// TIA Portal project "SORTIROZO_GEP_VEZERLES" (V15)

(* hardware
DEVICE "S71500/ET200MP-Station_1"  S7-1500 station
   slot 0: "Profilschiene_0"  6ES7 590-1***0-0AA0
   slot 1: "PLC_1"  CPU 1511-1 PN  6ES7 511-1AK00-0AB0  V1.8
   slot 2: "AI 8xU/I/RTD/TC ST_1"  AI 8xU/I/RTD/TC ST  6ES7 531-7KF00-0AB0  V2.0
   slot 3: "AI 8xU/I/RTD/TC ST_2"  AI 8xU/I/RTD/TC ST  6ES7 531-7KF00-0AB0  V2.0
   slot 4: "AI 8xU/I/RTD/TC ST_3"  AI 8xU/I/RTD/TC ST  6ES7 531-7KF00-0AB0  V2.0
   slot 5: "AI 8xU/I/RTD/TC ST_4"  AI 8xU/I/RTD/TC ST  6ES7 531-7KF00-0AB0  V2.0
   slot 6: "DI 16x24VDC BA_1"  DI 16x24VDC BA  6ES7 521-1BH10-0AA0  V1.0
*)

// ===== PLC "PLC_1"  CPU 1511-1 PN =====

VAR_GLOBAL   // PLC tag table "Standard-Variablentabelle"
   "System_Byte" AT %MB1 : Byte;
   "FirstScan" AT %M1.0 : Bool;
   "DiagStatusUpdate" AT %M1.1 : Bool;
   "AlwaysTRUE" AT %M1.2 : Bool;
   "AlwaysFALSE" AT %M1.3 : Bool;
   "Clock_Byte" AT %MB0 : Byte;
   "Clock_10Hz" AT %M0.0 : Bool;
   "Clock_5Hz" AT %M0.1 : Bool;
   "Clock_2.5Hz" AT %M0.2 : Bool;
   "Clock_2Hz" AT %M0.3 : Bool;
   "Clock_1.25Hz" AT %M0.4 : Bool;
   "Clock_1Hz" AT %M0.5 : Bool;
   "Clock_0.625Hz" AT %M0.6 : Bool;
   "Clock_0.5Hz" AT %M0.7 : Bool;
END_VAR

VAR_GLOBAL   // PLC tag table "IO"
   "PART_SENSOR_BIT_0" AT %I0.0 : Bool;
   "PART_SENSOR_BIT_1" AT %I0.1 : Bool;
   "PART_SENSOR_BIT_2" AT %I0.2 : Bool;
   "PART_SENSOR_BIT_3" AT %I0.3 : Bool;
   "PART_CAPACITIVE_SENSOR" AT %I0.4 : Bool;
   "PART_INDUCTIVE_SENSOR" AT %I0.5 : Bool;
   "REFLECTIVE_SENSOR" AT %I0.6 : Bool;
   "MANUAL_SWITCH" AT %I0.7 : Bool;
   "AUTO_SWITCH" AT %I1.0 : Bool;
   "START_BUTTON" AT %I1.1 : Bool;
   "STOP_BUTTON" AT %I1.2 : Bool;
   "ROBOT_PART_PLACE_GRAB_DEDECTED" AT %I1.3 : Bool;
   "ROBOT_PART_PLACE_X_IS_MOVING" AT %I1.4 : Bool;
   "ROBOT_PART_PLACE_Z_IS_MOVING" AT %I1.5 : Bool;
   "ROBOT_PART_PLACE_IS_ROTATING" AT %I1.6 : Bool;
   "ROBOT_PART_PICK_GRAB_DEDECTED" AT %I1.7 : Bool;
   "ROBOT_PART_PICK_X_IS_MOVING" AT %I2.0 : Bool;
   "ROBOT_PART_PICK_Z_IS_MOVING" AT %I2.1 : Bool;
   "ROBOT_PART_PICK_IS_ROTATING" AT %I2.2 : Bool;
   "STACK_LIGHT_RED" AT %Q0.0 : Bool;
   "STACK_LIGHT_GREEN" AT %Q0.1 : Bool;
   "STACK_LIGHT_YELLOW" AT %Q0.2 : Bool;
   "START_BUTTON_LIGHT" AT %Q0.3 : Bool;
   "STOP_BUTTON_LIGHT" AT %Q0.4 : Bool;
   "PART_INSPECT_STOP_BLADE" AT %Q0.5 : Bool;
   "PART_PICKUP_STOP_BLADE" AT %Q0.6 : Bool;
   "ROBOT_PART_PLACE_X" AT %Q0.7 : Bool;
   "ROBOT_PART_PLACE_Z" AT %Q1.0 : Bool;
   "ROBOT_PART_PLACE_GRAB" AT %Q1.1 : Bool;
   "ROBOT_PART_PLACE_ROTATE_CW" AT %Q1.2 : Bool;
   "ROBOT_PART_PLACE_ROTATE_CCW" AT %Q1.3 : Bool;
   "ROBOT_PART_PICK_X" AT %Q1.4 : Bool;
   "ROBOT_PART_PICK_Z" AT %Q1.5 : Bool;
   "ROBOT_PART_PICK_GRAB" AT %Q1.6 : Bool;
   "ROBOT_PART_PICK_ROTATE_CW" AT %Q1.7 : Bool;
   "ROBOT_PART_PICK_ROTATE_CCW" AT %Q2.0 : Bool;
   "PART_CONVEYOR" AT %Q2.1 : Bool;
END_VAR

DATA_BLOCK "mainProgram_DB"   // DB1
{ S7_Optimized_Access := 'TRUE' }
VERSION : 0.1
// stored: InstanceOfName mainProgram
"mainProgram"
BEGIN
END_DATA_BLOCK

DATA_BLOCK "mainProgram_DB_1"   // DB5
{ S7_Optimized_Access := 'TRUE' }
VERSION : 0.1
// stored: InstanceOfName mainProgram
"mainProgram"
BEGIN
END_DATA_BLOCK

// folder: System blocks/Program resources

DATA_BLOCK "IEC_Timer_0_DB"   // DB10
{ S7_Optimized_Access := 'TRUE' }
AUTHOR : Simatic
FAMILY : IEC
NAME : IEC_TMR
VERSION : 1.0
// stored: InstanceOfName IEC_TIMER
"IEC_TIMER"
BEGIN
END_DATA_BLOCK

// folder: (top level)

FUNCTION_BLOCK "mainProgram"   // FB1, SCL
{ S7_Optimized_Access := 'TRUE' }
VERSION : 0.1
   VAR_INPUT
      partSensorBit0 : Bool;
      partSensorBit1 : Bool;
      partSensorBit2 : Bool;
      partSensorBit3 : Bool;
      partCapacitiveSensor : Bool;
      partInductiveSensor : Bool;
      partReflectiveSensor : Bool;
      manualSwitch : Bool;
      autoSwitch : Bool;
      startButton : Bool;
      stopButton : Bool;
      robotPartPlaceGrabDedected : Bool;
      robotPartPlaceXIsMoving : Bool;
      robotPartPlaceZIsMoving : Bool;
      robotPartPlaceIsRotating : Bool;
      robotPartPickIsDedected : Bool;
      robotPartPickXIsMoving : Bool;
      robotPartPickZIsMoving : Bool;
      robotPartPickIsRotating : Bool;
   END_VAR
   VAR_OUTPUT
      stackLightRed : Bool;
      stackLightGreen : Bool;
      stackLightYellow : Bool;
      startButtonLighgt : Bool;
      stopButtonLight : Bool;
      partInspectStopBlade : Bool;
      partPickupStopBlade : Bool;
      robotPartPlaceX : Bool;
      robotPartPlaceZ : Bool;
      robotPartPlaceGrab : Bool;
      robotPartPlaceRotateCW : Bool;
      robotPartPlaceRotateCCW : Bool;
      robotPartPickX : Bool;
      robotPartPickZ : Bool;
      robotPartPickGrab : Bool;
      robotPartPickRotateCW : Bool;
      robotPartPickRotateCCW : Bool;
      partConveyor : Bool;
   END_VAR
   VAR
      robotRotateCounter : Int;
      "timer" : Time;
      onDelayCheck : Bool;
      fallingEgdeDedect : Bool;
      risingEgdeDedect : Bool;
      deviceState : Int;
      pickUpRobotState : Int;
      partPlaceRobotState : Int;
      cameraControlState : Int;
      partCameraData : Int;
      conveyorControlState : Int;
   END_VAR
   VAR CONSTANT
      CONVEYOR_MOVING_GRAY : Time := T#10s;
      CONVEYOR_MOVING_BLUE : Time := T#6s;
      ROBOT_PICK_NEXT_STEP_WAIT_TIME : Time := T#1s;
      STATE_INIT : Int;
      STATE_WAIT_FOR_START : Int := 1;
      STATE_IDLE : Int := 3;
      STATE_ROBOT_PICK_IDLE : Int;
      STATE_ROBOT_PICK_MOVE_PART_X : Int := 2;
      STATE_ROBOT_PICK_MOVE_PART_Z : Int := 3;
      STATE_ROBOT_PICK_GRAB_PART : Int := 4;
      STATE_ROBOT_PICK_ROTATE_TO_CONVEYER : Int := 7;
      STATE_ROBOT_PICK_PLACE_PART : Int := 8;
      STATE_ROBOT_PICK_CHECK_FOR_BASE_POSITION : Int := 9;
      STATE_CAMERA_IDLE : Int;
      STATE_CAMERA_READ_PRODUCT_DATA : Int := 1;
      STATE_CONVEYOR_IDLE : Int;
      STATE_CONVEYOR_GRAY : Int := 1;
      STATE_CONVEYOR_BLUE : Int := 2;
      STATE_CONVEYOR_GREEN : Int := 3;
      STATE_PART_PLACE_ROBOT_IDLE : Int;
      STATE_PART_PLACE_ROBOT_MOVE_X : Int := 1;
      STATE_PART_PLACE_ROBOT_MOVE_Z : Int := 2;
      STATE_PART_PLACE_ROBOT_GRAB : Int := 3;
      STATE_PART_PLACE_ROBOT_ROTATE_TO_CONVEYER : Int := 4;
      STATE_PART_PLACE_ROBOT_PLACE_PART : Int := 5;
   END_VAR
BEGIN
   CASE #deviceState OF
       #STATE_INIT:
           #stackLightYellow := "Clock_2Hz";
           #partInspectStopBlade := TRUE;
           #partPickupStopBlade := TRUE;
           #robotPartPlaceRotateCW := TRUE;

           "F_TRIG_DB"(CLK:=#robotPartPlaceIsRotating,
                       Q=>#fallingEgdeDedect);

           IF #fallingEgdeDedect THEN
               #stackLightYellow := FALSE;
               #stackLightRed := TRUE;
               #deviceState := #STATE_WAIT_FOR_START;
           END_IF;

       #STATE_WAIT_FOR_START:
           "R_TRIG_DB"(CLK:=#startButton,
                       Q=>#risingEgdeDedect);

           IF #risingEgdeDedect THEN
               #deviceState := #STATE_IDLE;
               #pickUpRobotState := #STATE_ROBOT_PICK_MOVE_PART_X;
           END_IF;
   END_CASE;

   CASE #pickUpRobotState OF
       #STATE_ROBOT_PICK_MOVE_PART_X:
           #robotPartPickX := TRUE;

           "F_TRIG_DB_1"(CLK:=#robotPartPickXIsMoving,
                         Q=>#fallingEgdeDedect);

           IF #fallingEgdeDedect THEN
               #pickUpRobotState := #STATE_ROBOT_PICK_MOVE_PART_Z;
           END_IF;

       #STATE_ROBOT_PICK_MOVE_PART_Z:
           #robotPartPickZ := TRUE;

           "F_TRIG_DB_2"(CLK:=#robotPartPickZIsMoving,
                         Q=>#fallingEgdeDedect);

           IF #fallingEgdeDedect THEN
               WAIT(WT := 10000);
               #robotPartPickGrab := TRUE;
               #stackLightRed := FALSE;
               #pickUpRobotState := #STATE_ROBOT_PICK_GRAB_PART;
           END_IF;

       #STATE_ROBOT_PICK_GRAB_PART:
           #robotPartPickGrab := TRUE;

           IF #robotPartPickIsDedected THEN
               WAIT(WT := 1000);
               #robotPartPickZ := FALSE;
               #pickUpRobotState := #STATE_ROBOT_PICK_ROTATE_TO_CONVEYER;
           END_IF;

       #STATE_ROBOT_PICK_ROTATE_TO_CONVEYER:
           #robotPartPickRotateCCW := TRUE;

           "F_TRIG_DB_3"(CLK:=#robotPartPickIsRotating,
                         Q=>#fallingEgdeDedect);

           IF #fallingEgdeDedect THEN
               WAIT(WT := 10000);
               #robotPartPickRotateCCW := FALSE;
               #pickUpRobotState := #STATE_ROBOT_PICK_PLACE_PART;
           END_IF;

       #STATE_ROBOT_PICK_PLACE_PART:
           #robotPartPickZ := TRUE;

           "F_TRIG_DB_2"(CLK := #robotPartPickZIsMoving,
                         Q => #fallingEgdeDedect);

           IF #fallingEgdeDedect THEN
               WAIT(WT := 10000);
               #robotPartPickGrab := FALSE;
               #robotPartPickZ := FALSE;
               #robotPartPickX := FALSE;
               #robotPartPickRotateCW := TRUE;
               #pickUpRobotState := #STATE_ROBOT_PICK_CHECK_FOR_BASE_POSITION;
               #cameraControlState := #STATE_CAMERA_READ_PRODUCT_DATA;
           END_IF;

   END_CASE;

   CASE #cameraControlState OF
       #STATE_CAMERA_READ_PRODUCT_DATA:
           IF #partSensorBit0 = TRUE AND #partSensorBit3 = TRUE THEN
               #conveyorControlState := #STATE_CONVEYOR_GRAY;
               #cameraControlState := #STATE_CAMERA_IDLE;
           END_IF;

           IF #partSensorBit0 = TRUE AND #partSensorBit1 = TRUE THEN
               #conveyorControlState := #STATE_CONVEYOR_BLUE;
               #cameraControlState := #STATE_CAMERA_IDLE;
           END_IF;

           IF #partSensorBit1 = TRUE AND #partSensorBit2 = TRUE THEN
               #conveyorControlState := #STATE_CONVEYOR_GREEN;
               #cameraControlState := #STATE_CAMERA_IDLE;
           END_IF;
   END_CASE;

   CASE #conveyorControlState OF
       #STATE_CONVEYOR_GRAY:
           #partConveyor := TRUE;
           #partInspectStopBlade := FALSE;
           #partPickupStopBlade := FALSE;

           "IEC_Timer_0_DB".TON(IN:=TRUE,
                                PT:=#CONVEYOR_MOVING_GRAY,
                                Q=>#onDelayCheck,
                                ET=>#timer);

           IF #onDelayCheck THEN
               #robotPartPickRotateCW := FALSE;
               #conveyorControlState := #STATE_CONVEYOR_IDLE;
               #partConveyor := FALSE;
               "IEC_Timer_0_DB".TON(IN := FALSE,
                                    PT := #CONVEYOR_MOVING_GRAY,
                                    Q => #onDelayCheck,
                                    ET => #timer);
               #pickUpRobotState := #STATE_ROBOT_PICK_MOVE_PART_X;
           END_IF;

           #STATE_CONVEYOR_BLUE .. #STATE_CONVEYOR_GREEN:
           #partPickupStopBlade := TRUE;

           #partConveyor := TRUE;
           #partInspectStopBlade := FALSE;

           "IEC_Timer_0_DB".TON(IN := TRUE,
                                PT := #CONVEYOR_MOVING_BLUE,
                                Q => #onDelayCheck,
                                ET => #timer);

           IF #onDelayCheck THEN
               #robotPartPickRotateCW := FALSE;
               #conveyorControlState := #STATE_CONVEYOR_IDLE;
               #partConveyor := FALSE;
               "IEC_Timer_0_DB".TON(IN := FALSE,
                                    PT := #CONVEYOR_MOVING_BLUE,
                                    Q => #onDelayCheck,
                                    ET => #timer);

               #partPlaceRobotState := #STATE_PART_PLACE_ROBOT_MOVE_X;
           END_IF;
   END_CASE;

   CASE #partPlaceRobotState OF
       #STATE_PART_PLACE_ROBOT_MOVE_X:
           #robotPartPlaceX := TRUE;

           "F_TRIG_DB_4"(CLK:=#robotPartPlaceXIsMoving,
                         Q=>#fallingEgdeDedect);

           IF #fallingEgdeDedect THEN
               #partPlaceRobotState := #STATE_PART_PLACE_ROBOT_MOVE_Z;
           END_IF;

       #STATE_PART_PLACE_ROBOT_MOVE_Z:
           #robotPartPlaceZ := TRUE;

           "F_TRIG_DB_5"(CLK:=#robotPartPlaceZIsMoving,
                         Q=>#fallingEgdeDedect);

           IF #fallingEgdeDedect THEN
               #partPlaceRobotState := #STATE_PART_PLACE_ROBOT_GRAB;
           END_IF;

       #STATE_PART_PLACE_ROBOT_GRAB:
           #robotPartPlaceGrab := TRUE;

           IF #robotPartPlaceGrab THEN
               #robotPartPlaceZ := FALSE;
               #partPlaceRobotState := #STATE_PART_PLACE_ROBOT_ROTATE_TO_CONVEYER;
           END_IF;

       #STATE_PART_PLACE_ROBOT_ROTATE_TO_CONVEYER:
           CASE #robotRotateCounter OF
               0:
                   #robotPartPlaceRotateCW := TRUE;

                   "F_TRIG_DB_8"(CLK:=#robotPartPlaceIsRotating,
                                 Q=>#fallingEgdeDedect);

                   IF #fallingEgdeDedect THEN
                       #robotPartPlaceRotateCW := FALSE;
                       #robotRotateCounter := 1;
                   END_IF;
               1:
                   #robotPartPlaceRotateCW := TRUE;

                   "F_TRIG_DB_8"(CLK := #robotPartPlaceIsRotating,
                                 Q => #fallingEgdeDedect);

                   IF #fallingEgdeDedect THEN
                       #robotPartPlaceRotateCW := FALSE;
                       #robotRotateCounter := 0;
                   #partPlaceRobotState := #STATE_PART_PLACE_ROBOT_PLACE_PART;
                   END_IF;
           END_CASE;

       #STATE_PART_PLACE_ROBOT_PLACE_PART:
           #robotPartPlaceZ := TRUE;

           "F_TRIG_DB_7"(CLK:=#robotPartPlaceZIsMoving,
                         Q=>#fallingEgdeDedect);

           IF #fallingEgdeDedect THEN
               #robotPartPickGrab := FALSE;
               #robotPartPlaceZ := FALSE;
           END_IF;

   END_CASE;
END_FUNCTION_BLOCK

FUNCTION "MHJ-PLC-Lab-Function-S71500" : Void   // FC9000, SCL
{ S7_Optimized_Access := 'TRUE' }
VERSION : 0.1
   VAR_TEMP
      Value : Byte;
      ForCounter : Int;
   END_VAR
   VAR CONSTANT
      Value_01_DW : DWord := 16#1223_5486;
      Value_02_DW : DWord := 16#A6C9_D1F5;
   END_VAR
BEGIN

   #Value:=PEEK(area := 16#82,
        dbNumber := 0,
        byteOffset := 511);
   #Value := #Value + 1;

   POKE(area := 16#82,
        dbNumber := 0,
        byteOffset := 511,
        value := #Value);

   POKE(area := 16#82,
        dbNumber := 0,
        byteOffset := 1016,
        value := #Value_01_DW);
   POKE(area := 16#82,
        dbNumber := 0,
        byteOffset := 1020,
        value := #Value_02_DW);

   FOR #ForCounter := 0 TO 63 DO
       #Value:=PEEK(area := 16#1,
            dbNumber := 0,
            byteOffset := #ForCounter);
       POKE(area := 16#81,
            dbNumber := 0,
            byteOffset := #ForCounter,
            value := #Value);
   END_FOR;
   #Value := PEEK(area := 16#1,
                  dbNumber := 0,
                  byteOffset := 512);
   POKE(area := 16#82,
        dbNumber := 0,
        byteOffset := 512,
        value := #Value);
END_FUNCTION

ORGANIZATION_BLOCK "Main"   // OB1, FBD, ProgramCycle
TITLE = "Main Program Sweep (Cycle)"
{ S7_Optimized_Access := 'TRUE' }
VERSION : 0.1
   VAR_INPUT
      Initial_Call : Bool;   // Initial call of this OB
      Remanence : Bool;   // =True, if remanent data are available
   END_VAR
BEGIN

REGION Network 1
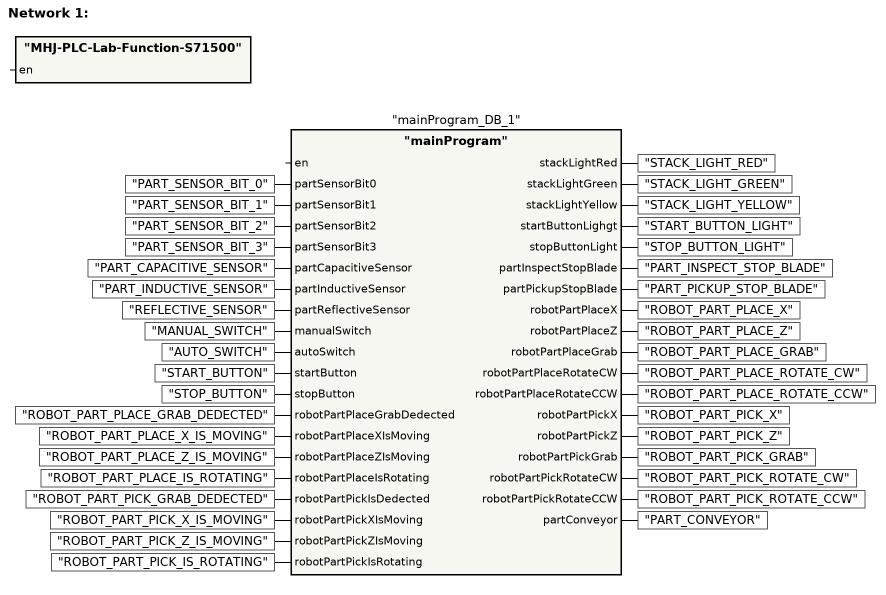
   "MHJ-PLC-Lab-Function-S71500"();
   "mainProgram_DB_1"(partSensorBit0 := "PART_SENSOR_BIT_0",   // "mainProgram"
                      partSensorBit1 := "PART_SENSOR_BIT_1",
                      partSensorBit2 := "PART_SENSOR_BIT_2",
                      partSensorBit3 := "PART_SENSOR_BIT_3",
                      partCapacitiveSensor := "PART_CAPACITIVE_SENSOR",
                      partInductiveSensor := "PART_INDUCTIVE_SENSOR",
                      partReflectiveSensor := "REFLECTIVE_SENSOR",
                      manualSwitch := "MANUAL_SWITCH",
                      autoSwitch := "AUTO_SWITCH",
                      startButton := "START_BUTTON",
                      stopButton := "STOP_BUTTON",
                      robotPartPlaceGrabDedected := "ROBOT_PART_PLACE_GRAB_DEDECTED",
                      robotPartPlaceXIsMoving := "ROBOT_PART_PLACE_X_IS_MOVING",
                      robotPartPlaceZIsMoving := "ROBOT_PART_PLACE_Z_IS_MOVING",
                      robotPartPlaceIsRotating := "ROBOT_PART_PLACE_IS_ROTATING",
                      robotPartPickIsDedected := "ROBOT_PART_PICK_GRAB_DEDECTED",
                      robotPartPickXIsMoving := "ROBOT_PART_PICK_X_IS_MOVING",
                      robotPartPickZIsMoving := "ROBOT_PART_PICK_Z_IS_MOVING",
                      robotPartPickIsRotating := "ROBOT_PART_PICK_IS_ROTATING",
                      stackLightRed => "STACK_LIGHT_RED",
                      stackLightGreen => "STACK_LIGHT_GREEN",
                      stackLightYellow => "STACK_LIGHT_YELLOW",
                      startButtonLighgt => "START_BUTTON_LIGHT",
                      stopButtonLight => "STOP_BUTTON_LIGHT",
                      partInspectStopBlade => "PART_INSPECT_STOP_BLADE",
                      partPickupStopBlade => "PART_PICKUP_STOP_BLADE",
                      robotPartPlaceX => "ROBOT_PART_PLACE_X",
                      robotPartPlaceZ => "ROBOT_PART_PLACE_Z",
                      robotPartPlaceGrab => "ROBOT_PART_PLACE_GRAB",
                      robotPartPlaceRotateCW => "ROBOT_PART_PLACE_ROTATE_CW",
                      robotPartPlaceRotateCCW => "ROBOT_PART_PLACE_ROTATE_CCW",
                      robotPartPickX => "ROBOT_PART_PICK_X",
                      robotPartPickZ => "ROBOT_PART_PICK_Z",
                      robotPartPickGrab => "ROBOT_PART_PICK_GRAB",
                      robotPartPickRotateCW => "ROBOT_PART_PICK_ROTATE_CW",
                      robotPartPickRotateCCW => "ROBOT_PART_PICK_ROTATE_CCW",
                      partConveyor => "PART_CONVEYOR");
END_REGION
END_ORGANIZATION_BLOCK